Fanuc KAREL source: kd00075.KL

-- PROVISIONAL review KL for V1013-1; original PC SHA256 262256b8e4447f336bef6d893fd44e883fb02d921c5ce3407a79073d84b7e12c
-- Incomplete behavior may be omitted. Consult companion uncertainty JSON. Do not deploy.
PROGRAM KD00075
%NOLOCKGROUP
VAR
  I : INTEGER
  J : INTEGER
  B : BOOLEAN
  R : REAL
  S : STRING[80]
BEGIN
  -- UNRESOLVED_PC offsets 5-24; opcodes 9D,81,18,9D,1B,9D,12,22,9D,13,04
  -- UNRESOLVED_PC offsets 29-33; opcodes 7F
END KD00075
